// TIA Portal V15.1 export
// export: Created 2024-05-17T05:38:22.718027Z, ExportSetting WithDefaults, DisplayName Totally Integrated Automation Portal, DisplayVersion V15.1 Update 5, DisplayName TIA Portal Openness, DisplayVersion V15.1 Update 5, DisplayName SINAMICS Startdrive Advanced, DisplayVersion V15.1, DisplayName G130, G150, S120, S150, SINAMICS MV, S210, DisplayVersion V15.1, DisplayName G110M, G120, G120C, G120D, G120P, DisplayVersion V15.1, DisplayName STEP 7 Professional, DisplayVersion V15.1 Update 5, DisplayName STEP 7 Safety, DisplayVersion V15.1, DisplayName WinCC Professional, DisplayVersion V15.1 Update 5, DisplayName SIMATIC Visualization Architect, DisplayVersion V15.1
DATA_BLOCK "_209230ZM01DataHandling"   // DB404
{ S7_Optimized_Access := 'FALSE' }
AUTHOR : VCC
VERSION : 0.1
// stored: AutoNumber false, DBAccessibleFromOPCUA true, IsOnlyStoredInLoadMemory false, IsWriteProtectedInAS false
   VAR RETAIN
      AC_209230NCB01VIDSMasterAlarm { ExternalAccessible := 'False'; ExternalVisible := 'False'; ExternalWritable := 'False'} : Bool;   // VIDS 209230NCB01 - Master Alarm
      AC_209230NCB01VIDSRFIDAlarm { ExternalAccessible := 'False'; ExternalVisible := 'False'; ExternalWritable := 'False'} : Bool;   // VIDS 209230NCB01 - RFID Alarm
      AC_209230NCB01VIDSTrackingAlarm { ExternalAccessible := 'False'; ExternalVisible := 'False'; ExternalWritable := 'False'} : Bool;   // VIDS 209230NCB01 - Tracking Alarm
      H_HMICmd : Word;   // Commands from HMI
      H_Anim : Word;   // Animation
      H_DBnr : Int;   // DB number
      H_209230NCB01TagSequenceIAnim : Word;   // Icon Animation
      H_HMI : Struct   // HMI Animation
         "209230NCB01VIDSMaster" : "H_HMI";   // HMI Animation
         "209230NCB01VIDSRFID" : "H_HMI";   // HMI Animation
         "209230NCB01VIDSTracking" : "H_HMI";   // HMI Animation
      END_STRUCT;
      H : Struct   // HMI Animation
         "209230NCB01VIDSMaster" : "H_LVIDSMaster";   // HMI Animation
         "209230NCB01VIDSRFID" : "H_LVIDSRFID";   // HMI Animation
         "209230NCB01VIDSTracking" : "H_LVIDSTrack";   // HMI Animation
      END_STRUCT;
      AlarmABCondition { ExternalAccessible := 'False'; ExternalVisible := 'False'; ExternalWritable := 'False'} : Bool;   // Alarm AB condition
      AlarmA { ExternalAccessible := 'False'; ExternalVisible := 'False'; ExternalWritable := 'False'} : Bool;   // Alarm A
      AlarmB { ExternalAccessible := 'False'; ExternalVisible := 'False'; ExternalWritable := 'False'} : Bool;   // Alarm B
      AlarmC { ExternalAccessible := 'False'; ExternalVisible := 'False'; ExternalWritable := 'False'} : Bool;   // Alarm C
      AlarmD { ExternalAccessible := 'False'; ExternalVisible := 'False'; ExternalWritable := 'False'} : Bool;   // Alarm D
      "209230NCB01TagSequence" { ExternalAccessible := 'False'; ExternalVisible := 'False'; ExternalWritable := 'False'} : "AlarmBits";   // Tag Sequence Alarm Bits
      "209230NCB01ReadBegin" { ExternalAccessible := 'False'; ExternalVisible := 'False'; ExternalWritable := 'False'} : Bool;   // Start Reading Body Data
      "209230NCB01BodyData" { ExternalAccessible := 'False'; ExternalVisible := 'False'; ExternalWritable := 'False'; S7_SetPoint := 'True'} : "VEMData";   // Body Data from VEMData
      "______209230NCB01_VIDS Master______" { ExternalAccessible := 'False'; ExternalVisible := 'False'; ExternalWritable := 'False'} : Bool;   // -----------------------------------------------------------------------------------
      "209230NCB01VIDS" { ExternalAccessible := 'False'; ExternalVisible := 'False'; ExternalWritable := 'False'; S7_SetPoint := 'True'} : "VIDS";   // Internal record
      "209230NCB01VEMData" { ExternalAccessible := 'False'; ExternalVisible := 'False'; ExternalWritable := 'False'; S7_SetPoint := 'True'} : "VEMData";   // VEM Data
      "209230NCB01VEMDataChange" { ExternalAccessible := 'False'; ExternalVisible := 'False'; ExternalWritable := 'False'; S7_SetPoint := 'True'} : "VEMData";   // VEM Data Change
      "209230NCB01VEMDataValid" { ExternalAccessible := 'False'; ExternalVisible := 'False'; ExternalWritable := 'False'; S7_SetPoint := 'True'} : Bool;   // VEM Data Valid
      "209230NCB01VEMDataNotValid" { ExternalAccessible := 'False'; ExternalVisible := 'False'; ExternalWritable := 'False'; S7_SetPoint := 'True'} : Bool;   // VEM Data Not Valid
      "209230NCB01GetVEMDataBusy" { ExternalAccessible := 'False'; ExternalVisible := 'False'; ExternalWritable := 'False'; S7_SetPoint := 'True'} : Bool;   // Get VEM Data Busy
      "209230NCB01MasterStatus" { ExternalAccessible := 'False'; ExternalVisible := 'False'; ExternalWritable := 'False'; S7_SetPoint := 'True'} : Int;   // Master - Status
      "______209230NCB01_VIDS RFID______" { ExternalAccessible := 'False'; ExternalVisible := 'False'; ExternalWritable := 'False'} : Bool;   // -----------------------------------------------------------------------------------
      "209230NCB01ReadOK" { ExternalAccessible := 'False'; ExternalVisible := 'False'; ExternalWritable := 'False'; S7_SetPoint := 'True'} : Bool;   // RFID - Read OK
      "209230NCB01ReadNOK" { ExternalAccessible := 'False'; ExternalVisible := 'False'; ExternalWritable := 'False'; S7_SetPoint := 'True'} : Bool;   // RFID - Read NOK
      "209230NCB01Busy" { ExternalAccessible := 'False'; ExternalVisible := 'False'; ExternalWritable := 'False'; S7_SetPoint := 'True'} : Bool;   // RFID - Busy
      "209230NCB01Status" { ExternalAccessible := 'False'; ExternalVisible := 'False'; ExternalWritable := 'False'; S7_SetPoint := 'True'} : Int;   // RFID - Status
      "______209230NCB01_VIDS Tracking______" { ExternalAccessible := 'False'; ExternalVisible := 'False'; ExternalWritable := 'False'} : Bool;   // -----------------------------------------------------------------------------------
      "209230NCB01TrackOK" { ExternalAccessible := 'False'; ExternalVisible := 'False'; ExternalWritable := 'False'; S7_SetPoint := 'True'} : Bool;   // Track - OK
      "209230NCB01TrackNOK" { ExternalAccessible := 'False'; ExternalVisible := 'False'; ExternalWritable := 'False'; S7_SetPoint := 'True'} : Bool;   // Track - Nok
      "209230NCB01TrackBusy" { ExternalAccessible := 'False'; ExternalVisible := 'False'; ExternalWritable := 'False'; S7_SetPoint := 'True'} : Bool;   // Track - Busy
      "209230NCB01TrackStatus" { ExternalAccessible := 'False'; ExternalVisible := 'False'; ExternalWritable := 'False'; S7_SetPoint := 'True'} : Int;   // Track - Status
      "209230NCB01SpecificData" { ExternalAccessible := 'False'; ExternalVisible := 'False'; ExternalWritable := 'False'; S7_SetPoint := 'True'} : Array[0..7925] of Byte;   // Specific Data Received
   END_VAR
BEGIN
END_DATA_BLOCK
